FUNCTION_BLOCK SampleSequencer EXTENDS TcoSequence
VAR_INPUT
END_VAR
VAR_OUTPUT
END_VAR
VAR
END_VAR

END_FUNCTION_BLOCK

(* stored: Version 1.1.0.1, ProductVersion 3.1.4024.12
   POU SampleSequencer: Id {162cfba3-e6ba-0cf8-16c6-2910ec4c4593}, SpecialFunc None *)
